// TIA Portal V16 export
// export: Created 2022-09-01T13:58:53.4848686Z, ExportSetting WithDefaults, DisplayName Totally Integrated Automation Portal, DisplayVersion V16, DisplayName TIA Portal Version Control Interface, DisplayVersion V16, DisplayName TIA Portal Openness, DisplayVersion V16, DisplayName STEP 7 Professional, DisplayVersion V16, DisplayName STEP 7 Safety, DisplayVersion V16, DisplayName WinCC Advanced, DisplayVersion V16
FUNCTION "Ciclo_Hórario_Filtros" : Void   // FC16, LAD
{ S7_Optimized_Access := 'TRUE' }
VERSION : 0.1
// stored: AutoNumber true, IsIECCheckEnabled false, SetENOAutomatically false, UDAEnableTagReadback false
   VAR_TEMP   // added for the SCL form of the ladder/FBD networks
      _w1 : Bool;
   END_VAR
BEGIN

REGION Network 1: Leitura de tempo do sistema
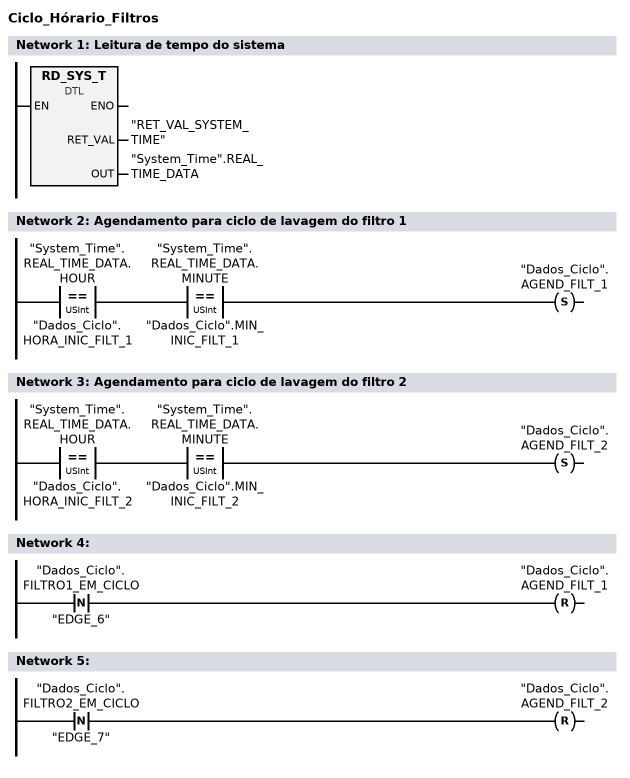
   RUNG wire#powerrail
      { S7_Templates := "date_type := DTL" } RD_SYS_T(RET_VAL => "RET_VAL_SYSTEM_TIME", OUT => "System_Time".REAL_TIME_DATA)
   END_RUNG
   // the same network as SCL:
   "RET_VAL_SYSTEM_TIME" := RD_SYS_T(OUT => "System_Time".REAL_TIME_DATA);
END_REGION

REGION Network 2: Agendamento para ciclo de lavagem do filtro 1
   RUNG wire#powerrail
      { S7_Templates := "SrcType := USInt" } EQ_Contact(in1 := "System_Time".REAL_TIME_DATA.HOUR, in2 := "Dados_Ciclo".HORA_INIC_FILT_1)
      { S7_Templates := "SrcType := USInt" } EQ_Contact(in1 := "System_Time".REAL_TIME_DATA.MINUTE, in2 := "Dados_Ciclo".MIN_INIC_FILT_1)
      S_Coil( "Dados_Ciclo".AGEND_FILT_1 )
   END_RUNG
   // the same network as SCL:
   IF ("System_Time".REAL_TIME_DATA.HOUR = "Dados_Ciclo".HORA_INIC_FILT_1) AND ("System_Time".REAL_TIME_DATA.MINUTE = "Dados_Ciclo".MIN_INIC_FILT_1) THEN
       "Dados_Ciclo".AGEND_FILT_1 := TRUE;
   END_IF;
END_REGION

REGION Network 3: Agendamento para ciclo de lavagem do filtro 2
   RUNG wire#powerrail
      { S7_Templates := "SrcType := USInt" } EQ_Contact(in1 := "System_Time".REAL_TIME_DATA.HOUR, in2 := "Dados_Ciclo".HORA_INIC_FILT_2)
      { S7_Templates := "SrcType := USInt" } EQ_Contact(in1 := "System_Time".REAL_TIME_DATA.MINUTE, in2 := "Dados_Ciclo".MIN_INIC_FILT_2)
      S_Coil( "Dados_Ciclo".AGEND_FILT_2 )
   END_RUNG
   // the same network as SCL:
   IF ("System_Time".REAL_TIME_DATA.HOUR = "Dados_Ciclo".HORA_INIC_FILT_2) AND ("System_Time".REAL_TIME_DATA.MINUTE = "Dados_Ciclo".MIN_INIC_FILT_2) THEN
       "Dados_Ciclo".AGEND_FILT_2 := TRUE;
   END_IF;
END_REGION

REGION Network 4
   RUNG wire#powerrail
      N_Contact(operand := "Dados_Ciclo".FILTRO1_EM_CICLO, bit := "EDGE_6")
      R_Coil( "Dados_Ciclo".AGEND_FILT_1 )
   END_RUNG
   // the same network as SCL:
   #_w1 := NOT "Dados_Ciclo".FILTRO1_EM_CICLO AND "EDGE_6";   // falling edge of "Dados_Ciclo".FILTRO1_EM_CICLO
   "EDGE_6" := "Dados_Ciclo".FILTRO1_EM_CICLO;
   IF #_w1 THEN "Dados_Ciclo".AGEND_FILT_1 := FALSE; END_IF;
END_REGION

REGION Network 5
   RUNG wire#powerrail
      N_Contact(operand := "Dados_Ciclo".FILTRO2_EM_CICLO, bit := "EDGE_7")
      R_Coil( "Dados_Ciclo".AGEND_FILT_2 )
   END_RUNG
   // the same network as SCL:
   #_w1 := NOT "Dados_Ciclo".FILTRO2_EM_CICLO AND "EDGE_7";   // falling edge of "Dados_Ciclo".FILTRO2_EM_CICLO
   "EDGE_7" := "Dados_Ciclo".FILTRO2_EM_CICLO;
   IF #_w1 THEN "Dados_Ciclo".AGEND_FILT_2 := FALSE; END_IF;
END_REGION
END_FUNCTION
